Universal Robots PolyScope program: external_control_with_onrobot_node.urp

Program external_control (installation=default directory=/programs createdIn=5.24.0 lastSavedIn=5.24.0 robotSerialNumber=20255201551)
Calibrated DH parameters: a=[0.000041, -0.099291, -0.571098, 0.00003, 0.000023, 0]; d=[0.180795, 429.375529, -433.059757, 3.858436, 0.11976, 0.115562]; alpha=[1.570181, -0.001408, 0.005532, 1.570403, -1.570135, 0]; deltaTheta=[0, -1.407965, 1.372291, 0.035675, 0, 0]
InitVariablesNode
Robot Program (runOnlyOnce=false)
  URCap RG Grip (OnRobot, OnRobot A/S) dataModel(rg-target-force=80.0, rg-target-width=0.09, Variable(key=on_return, variable(name=on_return)))
  URCap External Control (External Control, FZI Research Center for Information Technology)
